// TwinCAT 3 PLC project DCustomPLC
// Title: DMathCalculate
// Company: ITT_MathCalculate
// Author: Krishnpal
// ProjectVersion: 0.1.0.0
// Description: DynamicMathCalculate
// ProgramVersion: 3.1.4024.0
// libraries:
//   Tc2_Standard, * (Beckhoff Automation GmbH)
//   Tc2_System, * (Beckhoff Automation GmbH)
//   Tc3_Module, * (Beckhoff Automation GmbH)
// project tree:
//   POUs/ FB_Add.TcPOU (not stored), FB_Division.TcPOU (not stored), FB_Multiply.TcPOU (not stored), I_MathOperation.TcIO (not stored), MAIN.TcPOU (not stored)
//   Version/ Global_Version.TcGVL
//   VISUs/ PlcTask.TcTTO

CONFIGURATION DCustomPLC
    RESOURCE PLC ON TwinCAT3
        TASK PlcTask(INTERVAL := T#10ms, PRIORITY := 20);
        PROGRAM MAIN WITH PlcTask : MAIN;
    END_RESOURCE
END_CONFIGURATION

// ---- Version/Global_Version.TcGVL
{attribute 'TcGenerated'}
{attribute 'no-analysis'}
{attribute 'linkalways'}
// This function has been automatically generated from the project information.
VAR_GLOBAL CONSTANT
	{attribute 'const_non_replaced'}
	stLibVersion_DMathCalculate : ST_LibVersion := (iMajor := 0, iMinor := 1, iBuild := 0, iRevision := 0, nFlags := 0, sVersion := '0.1.0.0');
END_VAR
